// TIA Portal V18 export
DATA_BLOCK "PROCESS_DB"   // DB4
VERSION : 0.1
// stored: AutoNumber true, DBAccessibleFromOPCUA true, InstanceOfName PROCESS, InstanceOfType FB
"PROCESS"
   // VAR
   //    "RECUP TANK" { S7_SetPoint := 'True'} : "TANK";
   //    "HOT WATER TANK" { S7_SetPoint := 'True'} : "TANK";
   //    "CAUSTIC TANK" { S7_SetPoint := 'True'} : "TANK";
   //    "ACID TANK" { S7_SetPoint := 'True'} : "TANK";
   //    "RECUP PREP DONE" { S7_SetPoint := 'True'} : Bool;
   //    "HOT WTR PREP DONE" : Bool;
   //    "CAUSTIC PREP DONE" : Bool;
   //    "ACID PREP DONE" : Bool;
   //    "PREP FINISHED PULSE" : Bool;
   //    P1 : Bool;
   //    P2 : Bool;
   //    P3 : Bool;
   //    P4 : Bool;
   //    P5 : Bool;
   //    P6 : Bool;
   //    P7 : Bool;
   //    P8 : Bool;
   //    P9 : Bool;
   //    P10 : Bool;
   //    CIP_STARTED : Bool;
   //    "3 CIP FINISH PULSE" : Bool;
   //    "5 CIP FINISH PULSE" : Bool;
   //    "7 CIP FINISH PULSE" : Bool;
   //    "PUMP OK" : Bool;
   // END_VAR
   // VAR RETAIN
   //    "RECUP CIP DONE" : Array[0..4] of Bool;
   //    "HOT WTR CIP DONE" : Array[0..4] of Bool;
   //    "CAUSTIC CIP DONE" : Array[0..4] of Bool;
   //    "ACID CIP DONE" : Array[0..4] of Bool;
   //    "WATER FLUSH CIP DONE" : Array[0..4] of Bool;
   //    "CIP_STEP SELECTED" : Int;
   // END_VAR
   // VAR
   //    "CURCULATION PUMP" { S7_SetPoint := 'True'} : "PUMP";
   //    "BFV1 CTRL" { S7_SetPoint := 'True'} : "VALVE CTRL";
   //    "BFV2 CTRL" { S7_SetPoint := 'True'} : "VALVE CTRL";
   //    "BFV3 CTRL" { S7_SetPoint := 'True'} : "VALVE CTRL";
   //    "BFV4 CTRL" { S7_SetPoint := 'True'} : "VALVE CTRL";
   //    "BFV5 CTRL" { S7_SetPoint := 'True'} : "VALVE CTRL";
   //    "BFV6 CTRL" { S7_SetPoint := 'True'} : "VALVE CTRL";
   //    "BFV7 CTRL" { S7_SetPoint := 'True'} : "VALVE CTRL";
   //    "BFV8 CTRL" { S7_SetPoint := 'True'} : "VALVE CTRL";
   //    "BFV9 CTRL" { S7_SetPoint := 'True'} : "VALVE CTRL";
   //    "BFV10 CTRL" { S7_SetPoint := 'True'} : "VALVE CTRL";
   //    "BFV11 CTRL" { S7_SetPoint := 'True'} : "VALVE CTRL";
   //    "BFV12 CTRL" { S7_SetPoint := 'True'} : "VALVE CTRL";
   //    "BFV13 CTRL" { S7_SetPoint := 'True'} : "VALVE CTRL";
   //    "BFV14 CTRL" { S7_SetPoint := 'True'} : "VALVE CTRL";
   //    "BFV15 CTRL" { S7_SetPoint := 'True'} : "VALVE CTRL";
   //    "BFV16 CTRL" { S7_SetPoint := 'True'} : "VALVE CTRL";
   //    "BFV17 CTRL" { S7_SetPoint := 'True'} : "VALVE CTRL";
   //    "BFV18 CTRL" { S7_SetPoint := 'True'} : "VALVE CTRL";
   //    "BFV19 CTRL" { S7_SetPoint := 'True'} : "VALVE CTRL";
   //    "BFV20 CTRL" { S7_SetPoint := 'True'} : "VALVE CTRL";
   //    "CAUSTIC DOSING" { S7_SetPoint := 'True'} : "PUMP";
   //    "ACID DOSING" { S7_SetPoint := 'True'} : "PUMP";
   //    "RETURN PUMP 1" { S7_SetPoint := 'True'} : "PUMP";
   //    "RETURN PUMP 2" { S7_SetPoint := 'True'} : "PUMP";
   //    "RETURN PUMP 3" { S7_SetPoint := 'True'} : "PUMP";
   //    "WATER FLUSH" { S7_SetPoint := 'True'} : TON_TIME;
   // END_VAR
BEGIN
END_DATA_BLOCK
